Fanuc KAREL source: kt00381.KL

-- PROVISIONAL review KL for V770-1; original PC SHA256 eebdc7930ed6e5d6839efe875cfa2b8fced97b54888ed9986c633d793cfe9009
-- Incomplete behavior may be omitted. Consult companion uncertainty JSON. Do not deploy.
PROGRAM KT00381
%NOLOCKGROUP
VAR
  OUT : BOOLEAN
-- UNRESOLVED_DECL H1 type=002017
-- UNRESOLVED_DECL Y2 type=002018
BEGIN
  -- UNRESOLVED_PC offsets 5-19; opcodes 2E,22,9D,33,B4
  -- UNRESOLVED_PC offsets 24-38; opcodes 2E,22,9D,33,B2
  -- UNRESOLVED_PC offsets 43-68; opcodes 22,9D,33,B3,22,9D,33,B1,5A,23
  -- UNRESOLVED_PC offsets 73-77; opcodes 7F
END KT00381
